TYPE InputBase_8311D824 :
STRUCT
END_STRUCT
END_TYPE

(* stored: Version 1.2.0.0, ProductVersion 3.1.4024.11
   DUT InputBase_8311D824: Id {3dc656d2-8283-44cf-9cdd-94e74722da48} *)
